// TwinCAT 3 PLC project MCAG_PLC_Project
// ProgramVersion: 3.1.0.8
// libraries:
//   Tc2_MC2, * (Beckhoff Automation GmbH)
//   Tc2_Standard, * (Beckhoff Automation GmbH)
//   Tc2_System, * (Beckhoff Automation GmbH)
//   Tc3_Interfaces, * (Beckhoff Automation GmbH)
//   Tc3_Module, * (Beckhoff Automation GmbH)
// project tree:
//   DUTs/ DUT_AxisStatus_v0_01.TcDUT (not stored), DUT_AxisStatus_v0_02.TcDUT (not stored)
//   / PlcTask.TcTTO (not stored)
//   POUs/Hardware/EtherCAT_Terminals/Analog_Inputs/ FB_CalculateFrequency_3702_v0_01.TcPOU, FB_EL3702_v0_00.TcPOU (not stored), FB_EL3773_v0_00.TcPOU, FB_EL3773_v1_00.TcPOU (not stored)
//   POUs/Hardware/EtherCAT_Terminals/Digital_Inputs/ EL1002_v1_00.TcPOU, EL1004_v1_00.TcPOU (not stored), EL1008_v1_00.TcPOU, EL1012_v1_00.TcPOU (not stored), EL1014_v1_00.TcPOU, EL1018_v1_00.TcPOU, EL1024_v1_00.TcPOU, EL1034_v1_00.TcPOU, EL1084_v1_00.TcPOU (not stored), EL1088_v1_00.TcPOU (not stored), EL1094_v1_00.TcPOU (not stored), EL1098_v1_00.TcPOU, EL1104_v1_00.TcPOU, EL1114_v1_00.TcPOU (not stored), EL1124_v1_00.TcPOU, EL1134_v1_00.TcPOU (not stored), EL1144_v1_00.TcPOU (not stored), EL1202_v1_00.TcPOU, EL1252_v1_00.TcPOU (not stored), EL1258_v0_00.TcPOU, EL1259_v0_00.TcPOU, EL1262_v0_00.TcPOU, EL1502_v0_00.TcPOU (not stored), EL1512_v0_00.TcPOU, EL1702_v1_00.TcPOU, EL1712_v1_00.TcPOU, EL1722_v1_00.TcPOU, EL1804_v1_00.TcPOU (not stored), EL1808_v1_00.TcPOU (not stored), EL1809_v1_00.TcPOU, EL1814_v1_00.TcPOU (not stored), EL1819_v1_00.TcPOU (not stored), EL1859_v1_00.TcPOU (not stored), EL1862_v1_00.TcPOU, EL1872_v1_00.TcPOU (not stored), EL1889_v1_00.TcPOU, FB_EL1008_v1_00.TcPOU (not stored), FB_EL1202_v1_00.TcPOU (not stored), FB_EL1252ASM_v1_00.TcPOU, FB_EL1252_v1_00.TcPOU (not stored)
//   POUs/Hardware/EtherCAT_Terminals/Digital_Outputs/ EL2002_v1_00.TcPOU, EL2004_v1_00.TcPOU (not stored), EL2008_v1_00.TcPOU (not stored), EL2022_v1_00.TcPOU (not stored), EL2024_v1_00.TcPOU (not stored), EL2032_v1_00.TcPOU (not stored), EL2034_v1_00.TcPOU (not stored), EL2042_v1_00.TcPOU, EL2084_v1_00.TcPOU (not stored), EL2088_v1_00.TcPOU (not stored), EL2124_v1_00.TcPOU, EL2202_v0_00.TcPOU, EL2212_v0_00.TcPOU (not stored), EL2252_v0_00.TcPOU, EL2258_v0_00.TcPOU, EL2262_v0_00.TcPOU, EL2502_v0_00.TcPOU (not stored), EL2521_v1_00.TcPOU (not stored), EL2535_v0_00.TcPOU, FB_EL2008_v1_00.TcPOU
//   POUs/Hardware/EtherCAT_Terminals/Digital_Outputs/External_Types/ dutEL2521_Ctrl.TcDUT, dutEL2521_Status.TcDUT
//   POUs/Hardware/EtherCAT_Terminals/Digital_Outputs/Safety_Terminals/ EL1904_v0_00.TcPOU, EL1908_v0_00.TcPOU (not stored), EL2901_v0_00.TcPOU, EL2902_v0_00.TcPOU, EL2904_v0_00.TcPOU (not stored), EL2964_v0_00.TcPOU (not stored), EL6900_v0_00.TcPOU (not stored), FB_EL1904_v1_00.TcPOU (not stored), FB_EL2904_v1_00.TcPOU, FB_EL6900_v1_00.TcPOU
//   POUs/Hardware/EtherCAT_Terminals/Motion/ EL7211_v1_00.TcPOU, EL9576_v1_00.TcPOU
//   POUs/Hardware/EtherCAT_Terminals/System/ EL9505_V1_00.TcPOU
//   POUs/Hardware/Other/ EK1200.TcPOU
//   POUs/ MAIN.TcPOU
//   POUs/Motion/ FB_DriveVirtual.TcPOU, FB_NcAxis.TcPOU (not stored), FB_ReadParameterInNc.TcPOU (not stored), FB_SetPositionBiasInNc_v1_00.TcPOU (not stored), FB_SetPositionBiasInNc.TcPOU (not stored), FB_SetStateToBootstrapOnAX5000.TcPOU (not stored), FB_SetStateToInitOnAX5000.TcPOU (not stored), FB_SimulateEncoder.TcPOU (not stored), FB_WriteParameterInNc.TcPOU (not stored)

// ---- POUs/Hardware/EtherCAT_Terminals/Digital_Outputs/External_Types/dutEL2521_Ctrl.TcDUT
TYPE dutEL2521_Ctrl :
STRUCT
	///The control word (CW) is located in the output process image, and is transmitted from the controller to the terminal.
	///CW.0 FREQ_SEL 0bin / 1bin  Rapid change of the base frequency (only if the ramp function is inactive):
	///0bin = Base frequency 1 (object 8001:02)
	///1bin = Base frequency 2 (object 8001:03) 
	FREQ_SEL: BOOL;
	///CW.1 RAMP_DIS 1bin Operation of the ramp function is cancelled, in spite of object 8000:06 being active; if travel distance control is active, it is interrupted by this bit 
	RAMP_DIS: BOOL;
	///CW.2 GO_COUNTER 1bin  If travel distance control is active (object 8000:0A), then a pre-set counter value is approached when the bit is set 
	GO_COUNTER: BOOL;
	///CW.5 CNT_CLR 1bin The contents of the counter is cleared or set (object 8000:0B) by this bit. 
	///Any overflow or underflow bits that might be set are also cleared by this bit. 
	///The process can be edge triggered or level triggered (object 8000:05). 
	CNT_CLR: BOOL;
END_STRUCT
END_TYPE

// ---- POUs/Hardware/EtherCAT_Terminals/Digital_Outputs/External_Types/dutEL2521_Status.TcDUT
TYPE dutEL2521_Status :
STRUCT
	///The status word (SW) is located in the input process image, and is transmitted from the terminal to the controller.
	///SW.0 SEL_ACK/END_COUNTER 1bin  Confirms the change of base frequency. At activated travel distance control: target counter value reached 
	SEL_ACK: BOOL;
	///SW.1 RAMP_ACTIVE 1bin Ramp is currently being followed 
	RAMP_ACTIVE: BOOL;
	///SW.2 UNDERFLOW 1bin This bit is set if the 16-bit counter underflows (0 -> 65535). It is reset when the counter drops below two thirds of its measuring range (43690 -> 43689) or immediately an overflow occurs. 
	UNDERFLOW: BOOL;
	///SW.3 OVERFLOW 1bin This bit is set if the 16-bit counter overflows (65535 -> 0). It is reset when the counter exceeds one third of its measuring range (21845 -> 21846) or immediately an underflow occurs 
	OVERFLOW: BOOL;
	///SW.4 INPUT_T 1bin Status of INPUT_T 
	INPUT_T: BOOL;
	///SW.5 INPUT_Z 1bin Status of INPUT_Z 
	INPUT_Z: BOOL;
	///SW.6 ERROR 1bin General error bit, included with overflow/underflow 
	ERROR: BOOL;
END_STRUCT
END_TYPE

// ---- POUs/Hardware/EtherCAT_Terminals/Analog_Inputs/FB_CalculateFrequency_3702_v0_01.TcPOU
FUNCTION_BLOCK FB_CalculateFrequency_3702_v0_01
VAR CONSTANT
	///200 samples/period
	cBufferSize: INT := 1000;
END_VAR
VAR_INPUT
	En: BOOL;
	bCalculate: BOOL;
	aBufferValue: ARRAY[0..(cBuffersize - 1)] OF INT;
	aBufferDcTime: ARRAY[0..(cBuffersize - 1)] OF UDINT;
	///If curve has a DC offset
	nDCOffset: INT := 0;
END_VAR
VAR_OUTPUT
	EnO: BOOL;
	bError: BOOL;
	fActFrequency: LREAL;
END_VAR
VAR
	nIndex: INT;
	nFirstZeroCrossing: INT;
	nLastZeroCrossing: INT;
	rTimeFirst: REAL := 0;
	rTimeLast: REAL := 0;
	rTimeRes: REAL := 0;
	nCrossings: INT := 0;
END_VAR
VAR_TEMP
	rRange: REAL := 0;
	rTimeSpan: REAL := 0;
END_VAR

EnO:=En;
bError:=FALSE;
nCrossings:=0;
IF En AND bCalculate THEN
	//Serach for crossings of nDCOffset
	FOR nIndex:=1 TO cBuffersize-1 DO
		IF((aBufferValue[nIndex]>nDCOffset AND aBufferValue[nIndex-1]<=nDCOffset) OR (aBufferValue[nIndex]<nDCOffset AND aBufferValue[nIndex-1]>=nDCOffset))	THEN
			IF(nCrossings=0) THEN
				nFirstZeroCrossing:=nIndex;
			END_IF
			nLastZeroCrossing:=nIndex;
			nCrossings:=nCrossings+1;
		END_IF
	END_FOR	
	
	IF nFirstZeroCrossing < nLastZeroCrossing  AND  nCrossings>2 THEN
		//interpolate zero crossings for higher accuracy
		rTimeRes:=aBufferDcTime[1]-aBufferDcTime[0]; //Buffer must contain more than 2 values
		rRange:=INT_TO_REAL(ABS(aBufferValue[nFirstZeroCrossing-1]-aBufferValue[nFirstZeroCrossing]));
		rTimeFirst:=UDINT_TO_REAL( aBufferDcTime[nFirstZeroCrossing-1])+ABS(INT_TO_REAL(aBufferValue[nFirstZeroCrossing-1])/rRange*rTimeRes);
		rRange:=INT_TO_REAL(ABS(aBufferValue[nLastZeroCrossing-1]-aBufferValue[nLastZeroCrossing]));
		rTimeLast:=UDINT_TO_REAL( aBufferDcTime[nLastZeroCrossing-1])+ABS(INT_TO_REAL(aBufferValue[nLastZeroCrossing-1])/rRange*rTimeRes);

		//Time span first to last (considering that max one time counter overflow have occured in the total time range of the time buffer)	
		IF rTimeFirst<rTimeLast THEN		
			rTimeSpan:=rTimeLast-rTimeFirst;
		ELSE //overflow of counter once (only 32bit timestamp =4.29seconds)
			rTimeSpan:=4294967296.0-rTimeFirst+rTimeLast;
		END_IF
		
		fActFrequency:=1000000000.0/rTimeSpan*(nCrossings-1)/2; //two crossings per period => Average frequency over buffer.
	ELSE
		fActFrequency:=0;
	END_IF
END_IF

END_FUNCTION_BLOCK

// ---- POUs/Hardware/EtherCAT_Terminals/Analog_Inputs/FB_EL3773_v0_00.TcPOU
FUNCTION_BLOCK FB_EL3773_v0_00
VAR_INPUT
	En: BOOL;
END_VAR
VAR_OUTPUT
	EnO: BOOL;
	bL1Ok: BOOL;
	aL1Voltage: ARRAY[0..(cDcOversampling - 1)] OF INT;
	aL1Current: ARRAY[0..(cDcOversampling - 1)] OF INT;
	bL2Ok: BOOL;
	aL2Voltage: ARRAY[0..(cDcOversampling - 1)] OF INT;
	aL2Current: ARRAY[0..(cDcOversampling - 1)] OF INT;
	bL3Ok: BOOL;
	aL3Voltage: ARRAY[0..(cDcOversampling - 1)] OF INT;
	aL3Current: ARRAY[0..(cDcOversampling - 1)] OF INT;
	nDcTimeNextLatch: ULINT;
	bError: BOOL;
END_VAR
VAR
	L1_Voltage_Status_U1 AT %I*: UINT;
	L1_Voltage_Samples_U1_Samples AT %I*: ARRAY[0..(cDcOversampling - 1)] OF INT;
	L1_Current_Status_I1_Status AT %I*: UINT;
	L1_Current_Samples_I1_Samples AT %I*: ARRAY[0..(cDcOversampling - 1)] OF INT;
	L2_Voltage_Status_U2 AT %I*: UINT;
	L2_Voltage_Samples_U2_Samples AT %I*: ARRAY[0..(cDcOversampling - 1)] OF INT;
	L2_Current_Status_I2_Status AT %I*: UINT;
	L2_Current_Samples_I2_Samples AT %I*: ARRAY[0..(cDcOversampling - 1)] OF INT;
	L3_Voltage_Status_U3 AT %I*: UINT;
	L3_Voltage_Samples_U3_Samples AT %I*: ARRAY[0..(cDcOversampling - 1)] OF INT;
	L3_Current_Status_I3_Status AT %I*: UINT;
	L3_Current_Samples_I3_Samples AT %I*: ARRAY[0..(cDcOversampling - 1)] OF INT;
	AI_NextSync1Time_StartTimeNextLatch AT %I*: ULINT;
	WcState_WcState AT %I*: BOOL;
	InfoData_State AT %I*: UINT;
END_VAR

EnO:=En;

IF En AND (WcState_WcState OR InfoData_State<>16#8) THEN
	bError:=TRUE;
ELSE
	bError:=FALSE;
END_IF


IF En THEN
	IF bError=FALSE THEN
		IF (L1_Voltage_Status_U1 AND 2#0110000001000011)<>0
		OR (L1_Current_Status_I1_Status AND 2#0110000001000011)<>0 THEN
			bL1Ok:= FALSE;
		ELSE
			bL1Ok:= TRUE;
		END_IF
		
		IF (L2_Voltage_Status_U2 AND 2#0110000001000011)<>0
		OR (L2_Current_Status_I2_Status AND 2#0110000001000011)<>0 THEN
			bL2Ok:= FALSE;
		ELSE
			bL2Ok:= TRUE;
		END_IF
		
		IF (L3_Voltage_Status_U3 AND 2#0110000001000011)<>0
		OR (L3_Current_Status_I3_Status AND 2#0110000001000011)<>0 THEN
			bL3Ok:= FALSE;
		ELSE
			bL3Ok:= TRUE;
		END_IF

		IF bL1Ok THEN
			aL1Voltage:=L1_Voltage_Samples_U1_Samples;
			aL1Current:=L1_Current_Samples_I1_Samples;
		END_IF

		IF bL2Ok THEN
			aL2Voltage:=L2_Voltage_Samples_U2_Samples;
			aL2Current:=L2_Current_Samples_I2_Samples;
		END_IF

		IF bL3Ok THEN
			aL3Voltage:=L3_Voltage_Samples_U3_Samples;
			aL3Current:=L3_Current_Samples_I3_Samples;
		END_IF

		nDcTimeNextLatch:=AI_NextSync1Time_StartTimeNextLatch;
	ELSE
		bL1Ok:= FALSE;
		bL2Ok:= FALSE;
		bL3Ok:= FALSE;
		nDcTimeNextLatch:=0;
	END_IF
END_IF

END_FUNCTION_BLOCK

// ---- POUs/Hardware/EtherCAT_Terminals/Digital_Inputs/EL1002_v1_00.TcPOU
///EL1002 | 2-channel digital input terminal 24 V DC, 3 ms
FUNCTION_BLOCK EL1002_v1_00
VAR_INPUT
	En: BOOL;
END_VAR
VAR_OUTPUT
	EnO: BOOL;
	bDi_1: BOOL;
	bDi_2: BOOL;
	bError: BOOL;
END_VAR
VAR
	Channel_1_Input AT %I*: BOOL;
	Channel_2_Input AT %I*: BOOL;
	WcState_WcState AT %I*: BOOL;
	InfoData_State AT %I*: UINT;
END_VAR

EnO:=En;

IF En AND (WcState_WcState OR InfoData_State<>16#8) THEN
	bError:=TRUE;
ELSE
	bError:=FALSE;
END_IF

IF En THEN
	IF bError=FALSE THEN
		bDi_1:=Channel_1_Input;
		bDi_2:=Channel_2_Input;
	ELSE
		bDi_1:=FALSE;
		bDi_2:=FALSE;
	END_IF
END_IF

END_FUNCTION_BLOCK

// ---- POUs/Hardware/EtherCAT_Terminals/Digital_Inputs/EL1008_v1_00.TcPOU
///EL1008 | 8-channel digital input terminal 24 V DC, 3 ms
FUNCTION_BLOCK EL1008_v1_00
VAR_INPUT
	En: BOOL;
END_VAR
VAR_OUTPUT
	EnO: BOOL;
	bDi_1: BOOL;
	bDi_2: BOOL;
	bDi_3: BOOL;
	bDi_4: BOOL;
	bDi_5: BOOL;
	bDi_6: BOOL;
	bDi_7: BOOL;
	bDi_8: BOOL;
	bError: BOOL;
END_VAR
VAR
	Channel_1_Input AT %I*: BOOL;
	Channel_2_Input AT %I*: BOOL;
	Channel_3_Input AT %I*: BOOL;
	Channel_4_Input AT %I*: BOOL;
	Channel_5_Input AT %I*: BOOL;
	Channel_6_Input AT %I*: BOOL;
	Channel_7_Input AT %I*: BOOL;
	Channel_8_Input AT %I*: BOOL;
	WcState_WcState AT %I*: BOOL;
	InfoData_State AT %I*: UINT;
END_VAR

EnO:=En;

IF En AND (WcState_WcState OR InfoData_State<>16#8) THEN
	bError:=TRUE;
ELSE
	bError:=FALSE;
END_IF

IF En THEN
	IF bError=FALSE THEN
		bDi_1:=Channel_1_Input;
		bDi_2:=Channel_2_Input;
		bDi_3:=Channel_3_Input;
		bDi_4:=Channel_4_Input;
		bDi_5:=Channel_5_Input;
		bDi_6:=Channel_6_Input;
		bDi_7:=Channel_7_Input;
		bDi_8:=Channel_8_Input;
	ELSE
		bDi_1:=FALSE;
		bDi_2:=FALSE;
		bDi_3:=FALSE;
		bDi_4:=FALSE;
		bDi_5:=FALSE;
		bDi_6:=FALSE;
		bDi_7:=FALSE;
		bDi_8:=FALSE;
	END_IF
END_IF

END_FUNCTION_BLOCK

// ---- POUs/Hardware/EtherCAT_Terminals/Digital_Inputs/EL1014_v1_00.TcPOU
///EL1014 | 4-channel digital input terminal 24 V DC, 10 µs
FUNCTION_BLOCK EL1014_v1_00
VAR_INPUT
	En: BOOL;
END_VAR
VAR_OUTPUT
	EnO: BOOL;
	bDi_1: BOOL;
	bDi_2: BOOL;
	bDi_3: BOOL;
	bDi_4: BOOL;
	bError: BOOL;
END_VAR
VAR
	Channel_1_Input AT %I*: BOOL;
	Channel_2_Input AT %I*: BOOL;
	Channel_3_Input AT %I*: BOOL;
	Channel_4_Input AT %I*: BOOL;
	WcState_WcState AT %I*: BOOL;
	InfoData_State AT %I*: UINT;
END_VAR

EnO:=En;

IF En AND (WcState_WcState OR InfoData_State<>16#8) THEN
	bError:=TRUE;
ELSE
	bError:=FALSE;
END_IF

IF En THEN
	IF bError=FALSE THEN
		bDi_1:=Channel_1_Input;
		bDi_2:=Channel_2_Input;
		bDi_3:=Channel_3_Input;
		bDi_4:=Channel_4_Input;
	ELSE
		bDi_1:=FALSE;
		bDi_2:=FALSE;
		bDi_3:=FALSE;
		bDi_4:=FALSE;
	END_IF
END_IF

END_FUNCTION_BLOCK

// ---- POUs/Hardware/EtherCAT_Terminals/Digital_Inputs/EL1018_v1_00.TcPOU
///EL1018 | 8-channel digital input terminal 24 V DC, 10 µs
FUNCTION_BLOCK EL1018_v1_00
VAR_INPUT
	En: BOOL;
END_VAR
VAR_OUTPUT
	EnO: BOOL;
	bDi_1: BOOL;
	bDi_2: BOOL;
	bDi_3: BOOL;
	bDi_4: BOOL;
	bDi_5: BOOL;
	bDi_6: BOOL;
	bDi_7: BOOL;
	bDi_8: BOOL;
	bError: BOOL;
END_VAR
VAR
	Channel_1_Input AT %I*: BOOL;
	Channel_2_Input AT %I*: BOOL;
	Channel_3_Input AT %I*: BOOL;
	Channel_4_Input AT %I*: BOOL;
	Channel_5_Input AT %I*: BOOL;
	Channel_6_Input AT %I*: BOOL;
	Channel_7_Input AT %I*: BOOL;
	Channel_8_Input AT %I*: BOOL;
	WcState_WcState AT %I*: BOOL;
	InfoData_State AT %I*: UINT;
END_VAR

EnO:=En;

IF En AND (WcState_WcState OR InfoData_State<>16#8) THEN
	bError:=TRUE;
ELSE
	bError:=FALSE;
END_IF

IF En THEN
	IF bError=FALSE THEN
		bDi_1:=Channel_1_Input;
		bDi_2:=Channel_2_Input;
		bDi_3:=Channel_3_Input;
		bDi_4:=Channel_4_Input;
		bDi_5:=Channel_5_Input;
		bDi_6:=Channel_6_Input;
		bDi_7:=Channel_7_Input;
		bDi_8:=Channel_8_Input;
	ELSE
		bDi_1:=FALSE;
		bDi_2:=FALSE;
		bDi_3:=FALSE;
		bDi_4:=FALSE;
		bDi_5:=FALSE;
		bDi_6:=FALSE;
		bDi_7:=FALSE;
		bDi_8:=FALSE;
	END_IF
END_IF

END_FUNCTION_BLOCK

// ---- POUs/Hardware/EtherCAT_Terminals/Digital_Inputs/EL1024_v1_00.TcPOU
///EL1024 | 4-channel digital input terminal 24 V DC, 3 ms, for type 2 sensors
FUNCTION_BLOCK EL1024_v1_00
VAR_INPUT
	En: BOOL;
END_VAR
VAR_OUTPUT
	EnO: BOOL;
	bDi_1: BOOL;
	bDi_2: BOOL;
	bDi_3: BOOL;
	bDi_4: BOOL;
	bError: BOOL;
END_VAR
VAR
	Channel_1_Input AT %I*: BOOL;
	Channel_2_Input AT %I*: BOOL;
	Channel_3_Input AT %I*: BOOL;
	Channel_4_Input AT %I*: BOOL;
	WcState_WcState AT %I*: BOOL;
	InfoData_State AT %I*: UINT;
END_VAR

EnO:=En;

IF En AND (WcState_WcState OR InfoData_State<>16#8) THEN
	bError:=TRUE;
ELSE
	bError:=FALSE;
END_IF

IF En THEN
	IF bError=FALSE THEN
		bDi_1:=Channel_1_Input;
		bDi_2:=Channel_2_Input;
		bDi_3:=Channel_3_Input;
		bDi_4:=Channel_4_Input;
	ELSE
		bDi_1:=FALSE;
		bDi_2:=FALSE;
		bDi_3:=FALSE;
		bDi_4:=FALSE;
	END_IF
END_IF

END_FUNCTION_BLOCK

// ---- POUs/Hardware/EtherCAT_Terminals/Digital_Inputs/EL1034_v1_00.TcPOU
///EL1034 | 4-channel digital input terminal 24 V DC, 10 µs, potential-free inputs
FUNCTION_BLOCK EL1034_v1_00
VAR_INPUT
	En: BOOL;
END_VAR
VAR_OUTPUT
	EnO: BOOL;
	bDi_1: BOOL;
	bDi_2: BOOL;
	bDi_3: BOOL;
	bDi_4: BOOL;
	bError: BOOL;
END_VAR
VAR
	Channel_1_Input AT %I*: BOOL;
	Channel_2_Input AT %I*: BOOL;
	Channel_3_Input AT %I*: BOOL;
	Channel_4_Input AT %I*: BOOL;
	WcState_WcState AT %I*: BOOL;
	InfoData_State AT %I*: UINT;
END_VAR

EnO:=En;

IF En AND (WcState_WcState OR InfoData_State<>16#8) THEN
	bError:=TRUE;
ELSE
	bError:=FALSE;
END_IF

IF En THEN
	IF bError=FALSE THEN
		bDi_1:=Channel_1_Input;
		bDi_2:=Channel_2_Input;
		bDi_3:=Channel_3_Input;
		bDi_4:=Channel_4_Input;
	ELSE
		bDi_1:=FALSE;
		bDi_2:=FALSE;
		bDi_3:=FALSE;
		bDi_4:=FALSE;
	END_IF
END_IF

END_FUNCTION_BLOCK

// ---- POUs/Hardware/EtherCAT_Terminals/Digital_Inputs/EL1098_v1_00.TcPOU
///EL1098 | 8-channel digital input terminal 24 V DC, 10 µs, switching to negative potential
FUNCTION_BLOCK EL1098_v1_00
VAR_INPUT
	En: BOOL;
END_VAR
VAR_OUTPUT
	EnO: BOOL;
	bDi_1: BOOL;
	bDi_2: BOOL;
	bDi_3: BOOL;
	bDi_4: BOOL;
	bDi_5: BOOL;
	bDi_6: BOOL;
	bDi_7: BOOL;
	bDi_8: BOOL;
	bError: BOOL;
END_VAR
VAR
	Channel_1_Input AT %I*: BOOL;
	Channel_2_Input AT %I*: BOOL;
	Channel_3_Input AT %I*: BOOL;
	Channel_4_Input AT %I*: BOOL;
	Channel_5_Input AT %I*: BOOL;
	Channel_6_Input AT %I*: BOOL;
	Channel_7_Input AT %I*: BOOL;
	Channel_8_Input AT %I*: BOOL;
	WcState_WcState AT %I*: BOOL;
	InfoData_State AT %I*: UINT;
END_VAR

EnO:=En;

IF En AND (WcState_WcState OR InfoData_State<>16#8) THEN
	bError:=TRUE;
ELSE
	bError:=FALSE;
END_IF

IF En THEN
	IF bError=FALSE THEN
		bDi_1:=Channel_1_Input;
		bDi_2:=Channel_2_Input;
		bDi_3:=Channel_3_Input;
		bDi_4:=Channel_4_Input;
		bDi_5:=Channel_5_Input;
		bDi_6:=Channel_6_Input;
		bDi_7:=Channel_7_Input;
		bDi_8:=Channel_8_Input;
	ELSE
		bDi_1:=FALSE;
		bDi_2:=FALSE;
		bDi_3:=FALSE;
		bDi_4:=FALSE;
		bDi_5:=FALSE;
		bDi_6:=FALSE;
		bDi_7:=FALSE;
		bDi_8:=FALSE;
	END_IF
END_IF

END_FUNCTION_BLOCK

// ---- POUs/Hardware/EtherCAT_Terminals/Digital_Inputs/EL1104_v1_00.TcPOU
///EL1104 | 4-channel digital input terminals 24 V DC, 3 ms, 24 V and 0 V sensor supply
FUNCTION_BLOCK EL1104_v1_00
VAR_INPUT
	En: BOOL;
END_VAR
VAR_OUTPUT
	EnO: BOOL;
	bDi_1: BOOL;
	bDi_2: BOOL;
	bDi_3: BOOL;
	bDi_4: BOOL;
	bError: BOOL;
END_VAR
VAR
	Channel_1_Input AT %I*: BOOL;
	Channel_2_Input AT %I*: BOOL;
	Channel_3_Input AT %I*: BOOL;
	Channel_4_Input AT %I*: BOOL;
	WcState_WcState AT %I*: BOOL;
	InfoData_State AT %I*: UINT;
END_VAR

EnO:=En;

IF En AND (WcState_WcState OR InfoData_State<>16#8) THEN
	bError:=TRUE;
ELSE
	bError:=FALSE;
END_IF

IF En THEN
	IF bError=FALSE THEN
		bDi_1:=Channel_1_Input;
		bDi_2:=Channel_2_Input;
		bDi_3:=Channel_3_Input;
		bDi_4:=Channel_4_Input;
	ELSE
		bDi_1:=FALSE;
		bDi_2:=FALSE;
		bDi_3:=FALSE;
		bDi_4:=FALSE;
	END_IF
END_IF

END_FUNCTION_BLOCK

// ---- POUs/Hardware/EtherCAT_Terminals/Digital_Inputs/EL1124_v1_00.TcPOU
///EL1124 | 4-channel digital input terminal 5 V DC, 0.5 µs
FUNCTION_BLOCK EL1124_v1_00
VAR_INPUT
	En: BOOL;
END_VAR
VAR_OUTPUT
	EnO: BOOL;
	bDi_1: BOOL;
	bDi_2: BOOL;
	bDi_3: BOOL;
	bDi_4: BOOL;
	bError: BOOL;
END_VAR
VAR
	Channel_1_Input AT %I*: BOOL;
	Channel_2_Input AT %I*: BOOL;
	Channel_3_Input AT %I*: BOOL;
	Channel_4_Input AT %I*: BOOL;
	WcState_WcState AT %I*: BOOL;
	InfoData_State AT %I*: UINT;
END_VAR

EnO:=En;

IF En AND (WcState_WcState OR InfoData_State<>16#8) THEN
	bError:=TRUE;
ELSE
	bError:=FALSE;
END_IF

IF En THEN
	IF bError=FALSE THEN
		bDi_1:=Channel_1_Input;
		bDi_2:=Channel_2_Input;
		bDi_3:=Channel_3_Input;
		bDi_4:=Channel_4_Input;
	ELSE
		bDi_1:=FALSE;
		bDi_2:=FALSE;
		bDi_3:=FALSE;
		bDi_4:=FALSE;
	END_IF
END_IF

END_FUNCTION_BLOCK

// ---- POUs/Hardware/EtherCAT_Terminals/Digital_Inputs/EL1202_v1_00.TcPOU
///EL1202 | XFC, 2-channel digital input terminal 24 V DC, TON/TOFF 1 µs
FUNCTION_BLOCK EL1202_v1_00
VAR_INPUT
	En: BOOL;
END_VAR
VAR_OUTPUT
	EnO: BOOL;
	bDi_1: BOOL;
	bDi_2: BOOL;
	bError: BOOL;
END_VAR
VAR
	Channel_1_Input AT %I*: BOOL;
	Channel_2_Input AT %I*: BOOL;
	WcState_WcState AT %I*: BOOL;
	InfoData_State AT %I*: UINT;
END_VAR

EnO:=En;

IF En AND (WcState_WcState OR InfoData_State<>16#8) THEN
	bError:=TRUE;
ELSE
	bError:=FALSE;
END_IF

IF En THEN
	IF bError=FALSE THEN
		bDi_1:=Channel_1_Input;
		bDi_2:=Channel_2_Input;
	ELSE
		bDi_1:=FALSE;
		bDi_2:=FALSE;
	END_IF
END_IF

END_FUNCTION_BLOCK

// ---- POUs/Hardware/EtherCAT_Terminals/Digital_Inputs/EL1258_v0_00.TcPOU
///EL1258 | XFC, 8-channel digital input terminal with time stamp
FUNCTION_BLOCK EL1258_v0_00

END_FUNCTION_BLOCK

// ---- POUs/Hardware/EtherCAT_Terminals/Digital_Inputs/EL1259_v0_00.TcPOU
///EL1259 | XFC, 8-channel digital input + 8-channel digital output with Time-Stamp
FUNCTION_BLOCK EL1259_v0_00

END_FUNCTION_BLOCK

// ---- POUs/Hardware/EtherCAT_Terminals/Digital_Inputs/EL1262_v0_00.TcPOU
///EL1262 | XFC, 2-channel digital input terminal with oversampling
FUNCTION_BLOCK EL1262_v0_00

END_FUNCTION_BLOCK

// ---- POUs/Hardware/EtherCAT_Terminals/Digital_Inputs/EL1512_v0_00.TcPOU
///EL1512 | 2-channel, up/down counter, 24 V DC, 1 kHz, 16 bit
FUNCTION_BLOCK EL1512_v0_00

END_FUNCTION_BLOCK

// ---- POUs/Hardware/EtherCAT_Terminals/Digital_Inputs/EL1702_v1_00.TcPOU
///EL1702 | 2-channel digital input terminals 120V/230V AC, 10ms
FUNCTION_BLOCK EL1702_v1_00
VAR_INPUT
	En: BOOL;
END_VAR
VAR_OUTPUT
	EnO: BOOL;
	bDi_1: BOOL;
	bDi_2: BOOL;
	bError: BOOL;
END_VAR
VAR
	Channel_1_Input AT %I*: BOOL;
	Channel_2_Input AT %I*: BOOL;
	WcState_WcState AT %I*: BOOL;
	InfoData_State AT %I*: UINT;
END_VAR

EnO:=En;

IF En AND (WcState_WcState OR InfoData_State<>16#8) THEN
	bError:=TRUE;
ELSE
	bError:=FALSE;
END_IF

IF En THEN
	IF bError=FALSE THEN
		bDi_1:=Channel_1_Input;
		bDi_2:=Channel_2_Input;
	ELSE
		bDi_1:=FALSE;
		bDi_2:=FALSE;
	END_IF
END_IF

END_FUNCTION_BLOCK

// ---- POUs/Hardware/EtherCAT_Terminals/Digital_Inputs/EL1712_v1_00.TcPOU
///EL1712 | 2-channel digital input terminals 120V AC/DC, 10ms
FUNCTION_BLOCK EL1712_v1_00
VAR_INPUT
	En: BOOL;
END_VAR
VAR_OUTPUT
	EnO: BOOL;
	bDi_1: BOOL;
	bDi_2: BOOL;
	bError: BOOL;
END_VAR
VAR
	Channel_1_Input AT %I*: BOOL;
	Channel_2_Input AT %I*: BOOL;
	WcState_WcState AT %I*: BOOL;
	InfoData_State AT %I*: UINT;
END_VAR

EnO:=En;

IF En AND (WcState_WcState OR InfoData_State<>16#8) THEN
	bError:=TRUE;
ELSE
	bError:=FALSE;
END_IF

IF En THEN
	IF bError=FALSE THEN
		bDi_1:=Channel_1_Input;
		bDi_2:=Channel_2_Input;
	ELSE
		bDi_1:=FALSE;
		bDi_2:=FALSE;
	END_IF
END_IF

END_FUNCTION_BLOCK

// ---- POUs/Hardware/EtherCAT_Terminals/Digital_Inputs/EL1722_v1_00.TcPOU
///EL1722 | 2-channel digital input terminals 120V/230V AC, 10ms, no power contacts
FUNCTION_BLOCK EL1722_v1_00
VAR_INPUT
	En: BOOL;
END_VAR
VAR_OUTPUT
	EnO: BOOL;
	bDi_1: BOOL;
	bDi_2: BOOL;
	bError: BOOL;
END_VAR
VAR
	Channel_1_Input AT %I*: BOOL;
	Channel_2_Input AT %I*: BOOL;
	WcState_WcState AT %I*: BOOL;
	InfoData_State AT %I*: UINT;
END_VAR

EnO:=En;

IF En AND (WcState_WcState OR InfoData_State<>16#8) THEN
	bError:=TRUE;
ELSE
	bError:=FALSE;
END_IF

IF En THEN
	IF bError=FALSE THEN
		bDi_1:=Channel_1_Input;
		bDi_2:=Channel_2_Input;
	ELSE
		bDi_1:=FALSE;
		bDi_2:=FALSE;
	END_IF
END_IF

END_FUNCTION_BLOCK

// ---- POUs/Hardware/EtherCAT_Terminals/Digital_Inputs/EL1809_v1_00.TcPOU
///EL1809 | HD EtherCAT Terminals, 16-channel digital input 24 V DC, 3 ms
FUNCTION_BLOCK EL1809_v1_00
VAR_INPUT
	En: BOOL;
END_VAR
VAR_OUTPUT
	EnO: BOOL;
	bDi_1: BOOL;
	bDi_2: BOOL;
	bDi_3: BOOL;
	bDi_4: BOOL;
	bDi_5: BOOL;
	bDi_6: BOOL;
	bDi_7: BOOL;
	bDi_8: BOOL;
	bDi_9: BOOL;
	bDi_10: BOOL;
	bDi_11: BOOL;
	bDi_12: BOOL;
	bDi_13: BOOL;
	bDi_14: BOOL;
	bDi_15: BOOL;
	bDi_16: BOOL;
	bError: BOOL;
END_VAR
VAR
	Channel_1_Input AT %I*: BOOL;
	Channel_2_Input AT %I*: BOOL;
	Channel_3_Input AT %I*: BOOL;
	Channel_4_Input AT %I*: BOOL;
	Channel_5_Input AT %I*: BOOL;
	Channel_6_Input AT %I*: BOOL;
	Channel_7_Input AT %I*: BOOL;
	Channel_8_Input AT %I*: BOOL;
	Channel_9_Input AT %I*: BOOL;
	Channel_10_Input AT %I*: BOOL;
	Channel_11_Input AT %I*: BOOL;
	Channel_12_Input AT %I*: BOOL;
	Channel_13_Input AT %I*: BOOL;
	Channel_14_Input AT %I*: BOOL;
	Channel_15_Input AT %I*: BOOL;
	Channel_16_Input AT %I*: BOOL;
	WcState_WcState AT %I*: BOOL;
	InfoData_State AT %I*: UINT;
END_VAR

EnO:=En;

IF En AND (WcState_WcState OR InfoData_State<>16#8) THEN
	bError:=TRUE;
ELSE
	bError:=FALSE;
END_IF

IF En THEN
	IF bError=FALSE THEN
		bDi_1:=Channel_1_Input;
		bDi_2:=Channel_2_Input;
		bDi_3:=Channel_3_Input;
		bDi_4:=Channel_4_Input;
		bDi_5:=Channel_5_Input;
		bDi_6:=Channel_6_Input;
		bDi_7:=Channel_7_Input;
		bDi_8:=Channel_8_Input;
		bDi_9:=Channel_9_Input;
		bDi_10:=Channel_10_Input;
		bDi_11:=Channel_11_Input;
		bDi_12:=Channel_12_Input;
		bDi_13:=Channel_13_Input;
		bDi_14:=Channel_14_Input;
		bDi_15:=Channel_15_Input;
		bDi_16:=Channel_16_Input;
	ELSE
		bDi_1:=FALSE;
		bDi_2:=FALSE;
		bDi_3:=FALSE;
		bDi_4:=FALSE;
		bDi_5:=FALSE;
		bDi_6:=FALSE;
		bDi_7:=FALSE;
		bDi_8:=FALSE;
		bDi_9:=FALSE;
		bDi_10:=FALSE;
		bDi_11:=FALSE;
		bDi_12:=FALSE;
		bDi_13:=FALSE;
		bDi_14:=FALSE;
		bDi_15:=FALSE;
		bDi_16:=FALSE;
	END_IF
END_IF

END_FUNCTION_BLOCK

// ---- POUs/Hardware/EtherCAT_Terminals/Digital_Inputs/EL1862_v1_00.TcPOU
///EL1862 | 16-channel digital input terminals 24 V DC, 3 ms, type 3, flat-ribbon cable connection
FUNCTION_BLOCK EL1862_v1_00
VAR_INPUT
	En: BOOL;
END_VAR
VAR_OUTPUT
	EnO: BOOL;
	bDi_1: BOOL;
	bDi_2: BOOL;
	bDi_3: BOOL;
	bDi_4: BOOL;
	bDi_5: BOOL;
	bDi_6: BOOL;
	bDi_7: BOOL;
	bDi_8: BOOL;
	bDi_9: BOOL;
	bDi_10: BOOL;
	bDi_11: BOOL;
	bDi_12: BOOL;
	bDi_13: BOOL;
	bDi_14: BOOL;
	bDi_15: BOOL;
	bDi_16: BOOL;
	bError: BOOL;
END_VAR
VAR
	Channel_1_Input AT %I*: BOOL;
	Channel_2_Input AT %I*: BOOL;
	Channel_3_Input AT %I*: BOOL;
	Channel_4_Input AT %I*: BOOL;
	Channel_5_Input AT %I*: BOOL;
	Channel_6_Input AT %I*: BOOL;
	Channel_7_Input AT %I*: BOOL;
	Channel_8_Input AT %I*: BOOL;
	Channel_9_Input AT %I*: BOOL;
	Channel_10_Input AT %I*: BOOL;
	Channel_11_Input AT %I*: BOOL;
	Channel_12_Input AT %I*: BOOL;
	Channel_13_Input AT %I*: BOOL;
	Channel_14_Input AT %I*: BOOL;
	Channel_15_Input AT %I*: BOOL;
	Channel_16_Input AT %I*: BOOL;
	WcState_WcState AT %I*: BOOL;
	InfoData_State AT %I*: UINT;
END_VAR

EnO:=En;

IF En AND (WcState_WcState OR InfoData_State<>16#8) THEN
	bError:=TRUE;
ELSE
	bError:=FALSE;
END_IF

IF En THEN
	IF bError=FALSE THEN
		bDi_1:=Channel_1_Input;
		bDi_2:=Channel_2_Input;
		bDi_3:=Channel_3_Input;
		bDi_4:=Channel_4_Input;
		bDi_5:=Channel_5_Input;
		bDi_6:=Channel_6_Input;
		bDi_7:=Channel_7_Input;
		bDi_8:=Channel_8_Input;
		bDi_9:=Channel_9_Input;
		bDi_10:=Channel_10_Input;
		bDi_11:=Channel_11_Input;
		bDi_12:=Channel_12_Input;
		bDi_13:=Channel_13_Input;
		bDi_14:=Channel_14_Input;
		bDi_15:=Channel_15_Input;
		bDi_16:=Channel_16_Input;
	ELSE
		bDi_1:=FALSE;
		bDi_2:=FALSE;
		bDi_3:=FALSE;
		bDi_4:=FALSE;
		bDi_5:=FALSE;
		bDi_6:=FALSE;
		bDi_7:=FALSE;
		bDi_8:=FALSE;
		bDi_9:=FALSE;
		bDi_10:=FALSE;
		bDi_11:=FALSE;
		bDi_12:=FALSE;
		bDi_13:=FALSE;
		bDi_14:=FALSE;
		bDi_15:=FALSE;
		bDi_16:=FALSE;
	END_IF
END_IF

END_FUNCTION_BLOCK

// ---- POUs/Hardware/EtherCAT_Terminals/Digital_Inputs/EL1889_v1_00.TcPOU
///EL1889 | HD EtherCAT Terminal, 16-channel digital input 24 V DC, 3 ms, 0 V (ground) switching
FUNCTION_BLOCK EL1889_v1_00
VAR_INPUT
	En: BOOL;
END_VAR
VAR_OUTPUT
	EnO: BOOL;
	bDi_1: BOOL;
	bDi_2: BOOL;
	bDi_3: BOOL;
	bDi_4: BOOL;
	bDi_5: BOOL;
	bDi_6: BOOL;
	bDi_7: BOOL;
	bDi_8: BOOL;
	bDi_9: BOOL;
	bDi_10: BOOL;
	bDi_11: BOOL;
	bDi_12: BOOL;
	bDi_13: BOOL;
	bDi_14: BOOL;
	bDi_15: BOOL;
	bDi_16: BOOL;
	bError: BOOL;
END_VAR
VAR
	Channel_1_Input AT %I*: BOOL;
	Channel_2_Input AT %I*: BOOL;
	Channel_3_Input AT %I*: BOOL;
	Channel_4_Input AT %I*: BOOL;
	Channel_5_Input AT %I*: BOOL;
	Channel_6_Input AT %I*: BOOL;
	Channel_7_Input AT %I*: BOOL;
	Channel_8_Input AT %I*: BOOL;
	Channel_9_Input AT %I*: BOOL;
	Channel_10_Input AT %I*: BOOL;
	Channel_11_Input AT %I*: BOOL;
	Channel_12_Input AT %I*: BOOL;
	Channel_13_Input AT %I*: BOOL;
	Channel_14_Input AT %I*: BOOL;
	Channel_15_Input AT %I*: BOOL;
	Channel_16_Input AT %I*: BOOL;
	WcState_WcState AT %I*: BOOL;
	InfoData_State AT %I*: UINT;
END_VAR

EnO:=En;

IF En AND (WcState_WcState OR InfoData_State<>16#8) THEN
	bError:=TRUE;
ELSE
	bError:=FALSE;
END_IF

IF En THEN
	IF bError=FALSE THEN
		bDi_1:=Channel_1_Input;
		bDi_2:=Channel_2_Input;
		bDi_3:=Channel_3_Input;
		bDi_4:=Channel_4_Input;
		bDi_5:=Channel_5_Input;
		bDi_6:=Channel_6_Input;
		bDi_7:=Channel_7_Input;
		bDi_8:=Channel_8_Input;
		bDi_9:=Channel_9_Input;
		bDi_10:=Channel_10_Input;
		bDi_11:=Channel_11_Input;
		bDi_12:=Channel_12_Input;
		bDi_13:=Channel_13_Input;
		bDi_14:=Channel_14_Input;
		bDi_15:=Channel_15_Input;
		bDi_16:=Channel_16_Input;
	ELSE
		bDi_1:=FALSE;
		bDi_2:=FALSE;
		bDi_3:=FALSE;
		bDi_4:=FALSE;
		bDi_5:=FALSE;
		bDi_6:=FALSE;
		bDi_7:=FALSE;
		bDi_8:=FALSE;
		bDi_9:=FALSE;
		bDi_10:=FALSE;
		bDi_11:=FALSE;
		bDi_12:=FALSE;
		bDi_13:=FALSE;
		bDi_14:=FALSE;
		bDi_15:=FALSE;
		bDi_16:=FALSE;
	END_IF
END_IF

END_FUNCTION_BLOCK

// ---- POUs/Hardware/EtherCAT_Terminals/Digital_Inputs/FB_EL1252ASM_v1_00.TcPOU
FUNCTION_BLOCK FB_EL1252ASM_v1_00
VAR_INPUT
	En: BOOL;
END_VAR
VAR_OUTPUT
	EnO: BOOL;
	Di_1: BOOL;
	Di_2: BOOL;
	Di_1_LatchTimePos: ULINT;
	Di_2_LatchTimePos: ULINT;
	Di_1_LatchTimeNeg: ULINT;
	Di_2_LatchTimeNeg: ULINT;
	///Below bits can be used but then they must be enabled in the COE of the card. Nicklas suggested to not use these (since something wss written that you then only were allowed to read the latch time onece (some kkind of auto reset??))	
	///Di_1_LatchNeg:BOOL;
	///	Di_1_LatchPos:BOOL;
	///	Di_2_LatchNeg:BOOL;
	///	Di_2_LatchPos:BOOL;
	Error: BOOL;
END_VAR
VAR
	Channel_1_Input AT %I*: BOOL;
	Channel_2_Input AT %I*: BOOL;
	///Latch_Status1 AT %I*: USINT;
	///	Latch_Status2 AT %I*: USINT;
	Latch_LatchPos1 AT %I*: ULINT;
	Latch_LatchNeg1 AT %I*: ULINT;
	Latch_LatchPos2 AT %I*: ULINT;
	Latch_LatchNeg2 AT %I*: ULINT;
	WcState_WcState AT %I*: BOOL;
	InfoData_State AT %I*: UINT;
END_VAR

EnO:=En;

IF En AND (WcState_WcState OR InfoData_State<>16#8) THEN //InfoData_State==0 => in OP mode
	Error:=TRUE;
ELSE
	Error:=FALSE;
END_IF

IF En THEN
	IF Error=FALSE THEN
		Di_1:=Channel_1_Input;
		Di_2:=Channel_2_Input;
	(*	Di_1_LatchPos:=Latch_Status1.0;
		Di_1_LatchNeg:=Latch_Status1.1;
		Di_2_LatchPos:=Latch_Status2.0;
		Di_2_LatchNeg:=Latch_Status2.1;*)
		Di_1_LatchTimePos:=Latch_LatchPos1;
		Di_2_LatchTimePos:=Latch_LatchPos2;		
		Di_1_LatchTimeNeg:=Latch_LatchNeg1;		
		Di_2_LatchTimeNeg:=Latch_LatchNeg2;
		
	ELSE
		Di_1:=FALSE;
		Di_2:=FALSE;
	END_IF
END_IF

END_FUNCTION_BLOCK

// ---- POUs/Hardware/EtherCAT_Terminals/Digital_Outputs/EL2002_v1_00.TcPOU
///EL2002 | 2-channel digital output terminal 24 V DC, 0.5 A
FUNCTION_BLOCK EL2002_v1_00
VAR_INPUT
	En: BOOL;
	bDo_1: BOOL;
	bDo_2: BOOL;
END_VAR
VAR_OUTPUT
	EnO: BOOL;
	bError: BOOL;
END_VAR
VAR
	Channel_1_Output AT %Q*: BOOL;
	Channel_2_Output AT %Q*: BOOL;
	WcState_WcState AT %I*: BOOL;
	InfoData_State AT %I*: UINT;
END_VAR

EnO:=En;

IF En AND (WcState_WcState OR InfoData_State<>16#8) THEN
	bError:=TRUE;
ELSE
	bError:=FALSE;
END_IF

IF En THEN
	IF bError=FALSE THEN
		Channel_1_Output:=bDo_1;
		Channel_2_Output:=bDo_2;
	END_IF
END_IF

END_FUNCTION_BLOCK

// ---- POUs/Hardware/EtherCAT_Terminals/Digital_Outputs/EL2042_v1_00.TcPOU
///EL2042 | 2-channel digital output terminal 24 V DC, 2 x 4 A/1 x 8 A
FUNCTION_BLOCK EL2042_v1_00
VAR_INPUT
	En: BOOL;
	bDo_1: BOOL;
	bDo_2: BOOL;
END_VAR
VAR_OUTPUT
	EnO: BOOL;
	bError: BOOL;
END_VAR
VAR
	Channel_1_Output AT %Q*: BOOL;
	Channel_2_Output AT %Q*: BOOL;
	WcState_WcState AT %I*: BOOL;
	InfoData_State AT %I*: UINT;
END_VAR

EnO:=En;

IF En AND (WcState_WcState OR InfoData_State<>16#8) THEN
	bError:=TRUE;
ELSE
	bError:=FALSE;
END_IF

IF En THEN
	IF bError=FALSE THEN
		Channel_1_Output:=bDo_1;
		Channel_2_Output:=bDo_2;
	END_IF
END_IF

END_FUNCTION_BLOCK

// ---- POUs/Hardware/EtherCAT_Terminals/Digital_Outputs/EL2124_v1_00.TcPOU
///EL2124 | 4-channel digital output terminal 5 V DC, 20 mA
FUNCTION_BLOCK EL2124_v1_00
VAR_INPUT
	En: BOOL;
	bDo_1: BOOL;
	bDo_2: BOOL;
	bDo_3: BOOL;
	bDo_4: BOOL;
END_VAR
VAR_OUTPUT
	EnO: BOOL;
	bError: BOOL;
END_VAR
VAR
	Channel_1_Output AT %Q*: BOOL;
	Channel_2_Output AT %Q*: BOOL;
	Channel_3_Output AT %Q*: BOOL;
	Channel_4_Output AT %Q*: BOOL;
	WcState_WcState AT %I*: BOOL;
	InfoData_State AT %I*: UINT;
END_VAR

EnO:=En;

IF En AND (WcState_WcState OR InfoData_State<>16#8) THEN
	bError:=TRUE;
ELSE
	bError:=FALSE;
END_IF

IF En THEN
	IF bError=FALSE THEN
		Channel_1_Output:=bDo_1;
		Channel_2_Output:=bDo_2;
		Channel_3_Output:=bDo_3;
		Channel_4_Output:=bDo_4;
	END_IF
END_IF

END_FUNCTION_BLOCK

// ---- POUs/Hardware/EtherCAT_Terminals/Digital_Outputs/EL2202_v0_00.TcPOU
///EL2202 | XFC, 2-channel digital output terminal 24 V DC, TON/TOFF 1 µs, push-pull outputs, tri-state
FUNCTION_BLOCK EL2202_v0_00

END_FUNCTION_BLOCK

// ---- POUs/Hardware/EtherCAT_Terminals/Digital_Outputs/EL2252_v0_00.TcPOU
///EL2252 | XFC, 2-channel digital output terminal with time stamp, tri-state
FUNCTION_BLOCK EL2252_v0_00

END_FUNCTION_BLOCK

// ---- POUs/Hardware/EtherCAT_Terminals/Digital_Outputs/EL2258_v0_00.TcPOU
///EL2258 | XFC, 8-channel digital output terminal with time stamp
FUNCTION_BLOCK EL2258_v0_00

END_FUNCTION_BLOCK

// ---- POUs/Hardware/EtherCAT_Terminals/Digital_Outputs/EL2262_v0_00.TcPOU
///EL2262 | XFC, 2-channel digital output terminal with oversampling
FUNCTION_BLOCK EL2262_v0_00

END_FUNCTION_BLOCK

// ---- POUs/Hardware/EtherCAT_Terminals/Digital_Outputs/EL2535_v0_00.TcPOU
///EL2535 | 2-channel pulse width current terminals 24 V DC
FUNCTION_BLOCK EL2535_v0_00

END_FUNCTION_BLOCK

// ---- POUs/Hardware/EtherCAT_Terminals/Digital_Outputs/FB_EL2008_v1_00.TcPOU
///EL2008 | 8-channel digital output terminal 24 V DC, 0.5 A
FUNCTION_BLOCK FB_EL2008_v1_00
VAR_INPUT
	En: BOOL;
	bDo_1: BOOL;
	bDo_2: BOOL;
	bDo_3: BOOL;
	bDo_4: BOOL;
	bDo_5: BOOL;
	bDo_6: BOOL;
	bDo_7: BOOL;
	bDo_8: BOOL;
END_VAR
VAR_OUTPUT
	EnO: BOOL;
	bError: BOOL;
END_VAR
VAR
	Channel_1_Output AT %Q*: BOOL;
	Channel_2_Output AT %Q*: BOOL;
	Channel_3_Output AT %Q*: BOOL;
	Channel_4_Output AT %Q*: BOOL;
	Channel_5_Output AT %Q*: BOOL;
	Channel_6_Output AT %Q*: BOOL;
	Channel_7_Output AT %Q*: BOOL;
	Channel_8_Output AT %Q*: BOOL;
	WcState_WcState AT %I*: BOOL;
	InfoData_State AT %I*: UINT;
END_VAR

EnO:=En;

IF En AND (WcState_WcState OR InfoData_State<>16#8) THEN
	bError:=TRUE;
ELSE
	bError:=FALSE;
END_IF

IF En THEN
	IF bError=FALSE THEN
		Channel_1_Output:=bDo_1;
		Channel_2_Output:=bDo_2;
		Channel_3_Output:=bDo_3;
		Channel_4_Output:=bDo_4;
		Channel_5_Output:=bDo_5;
		Channel_6_Output:=bDo_6;
		Channel_7_Output:=bDo_7;
		Channel_8_Output:=bDo_8;
	END_IF
END_IF

END_FUNCTION_BLOCK

// ---- POUs/Hardware/EtherCAT_Terminals/Digital_Outputs/Safety_Terminals/EL1904_v0_00.TcPOU
///EL1904 | 4-channel digital input terminal, TwinSAFE, 24 V DC
FUNCTION_BLOCK EL1904_v0_00

END_FUNCTION_BLOCK

// ---- POUs/Hardware/EtherCAT_Terminals/Digital_Outputs/Safety_Terminals/EL2901_v0_00.TcPOU
///EL2901 | Potential supply terminal, TwinSAFE, 24 V DC, 10 A
FUNCTION_BLOCK EL2901_v0_00

END_FUNCTION_BLOCK

// ---- POUs/Hardware/EtherCAT_Terminals/Digital_Outputs/Safety_Terminals/EL2902_v0_00.TcPOU
///EL2902 | 2-channel digital output terminal, TwinSAFE, 24 V DC, 2.3 A
FUNCTION_BLOCK EL2902_v0_00

END_FUNCTION_BLOCK

// ---- POUs/Hardware/EtherCAT_Terminals/Digital_Outputs/Safety_Terminals/FB_EL2904_v1_00.TcPOU
///EL2904 | 4-channel digital output terminal, TwinSAFE, 24 V DC, 0.5 A
FUNCTION_BLOCK FB_EL2904_v1_00
VAR_INPUT
	En: BOOL;
END_VAR
VAR_OUTPUT
	EnO: BOOL;
	bDo_1: BOOL;
	bDo_2: BOOL;
	bDo_3: BOOL;
	bDo_4: BOOL;
	bError: BOOL;
	sState: STRING;
	sDiag: STRING;
END_VAR
VAR
	Message_X_Info_Data_State AT %I*: USINT;
	Message_X_Info_Data_Diag AT %I*: USINT;
	Message_X_Output_Safe_Data AT %I*: BYTE;
	WcState_WcState AT %I*: BOOL;
	InfoData_State AT %I*: UINT;
END_VAR

EnO:=En;

IF En AND (WcState_WcState OR InfoData_State<>16#8) THEN
	bError:=TRUE;
ELSE
	bError:=FALSE;
END_IF

IF En THEN
	IF bError=FALSE THEN
		CASE Message_X_Info_Data_State OF
		0:
			sState:='Undefined';
		100:
			sState:='RESET';
		101:
			sState:='SESSION';
		102:
			sState:='CONNECTION';
		103:
			sState:='PARAMETER';
		104:
			sState:='DATA';
		105:
			sState:='SHUTDOWN';
		ELSE	
			sState:='Unknown';
		END_CASE

		sDiag:=USINT_TO_STRING(Message_X_Info_Data_Diag);

		bDo_1:=Message_X_Output_Safe_Data.0;
		bDo_2:=Message_X_Output_Safe_Data.1;
		bDo_3:=Message_X_Output_Safe_Data.2;
		bDo_4:=Message_X_Output_Safe_Data.3;
	ELSE
		sState:='';
		sDiag:='';

	END_IF
END_IF

END_FUNCTION_BLOCK

// ---- POUs/Hardware/EtherCAT_Terminals/Digital_Outputs/Safety_Terminals/FB_EL6900_v1_00.TcPOU
///EL6900 | TwinSAFE PLC
FUNCTION_BLOCK FB_EL6900_v1_00
VAR_INPUT
	En: BOOL;
END_VAR
VAR_OUTPUT
	EnO: BOOL;
	bError: BOOL;
END_VAR
VAR
	WcState_WcState AT %I*: BOOL;
	InfoData_State AT %I*: UINT;
END_VAR

EnO:=En;

IF En AND (WcState_WcState OR InfoData_State<>16#8) THEN
	bError:=TRUE;
ELSE
	bError:=FALSE;
END_IF

END_FUNCTION_BLOCK

// ---- POUs/Hardware/EtherCAT_Terminals/Motion/EL7211_v1_00.TcPOU
///EL7211 | Servo motor termional 5 A
FUNCTION_BLOCK EL7211_v1_00
VAR_INPUT
	En: BOOL;
END_VAR
VAR_OUTPUT
	EnO: BOOL;

	bError: BOOL;
END_VAR
VAR
	WcState_WcState AT %I*: BOOL;
	InfoData_State AT %I*: UINT;
END_VAR

EnO:=En;

IF En AND (WcState_WcState OR InfoData_State<>16#8) THEN
	bError:=TRUE;
ELSE
	bError:=FALSE;
END_IF

END_FUNCTION_BLOCK

// ---- POUs/Hardware/EtherCAT_Terminals/Motion/EL9576_v1_00.TcPOU
///EL9576 | Brake terminal (vap and resistor)
FUNCTION_BLOCK EL9576_v1_00
VAR_INPUT
	En: BOOL;
END_VAR
VAR_OUTPUT
	EnO: BOOL;
	bError: BOOL;	
	OverTemperature: BOOL;
	I2TError : BOOL;
	I2TWarning : BOOL;
	OverVoltage  : BOOL;
	UnderVoltage : BOOL;
	ChopperOn : BOOL;
	DCLinkVoltage : LREAL;
	DutyCycle  : LREAL;
	ResistorCurrent : LREAL;
	
END_VAR
VAR
	BCTOverTemperature AT %I*: BOOL;
	BCTI2TError AT %I*: BOOL;
	BCTI2TWarning AT %I*: BOOL;
	BCTOverVoltage  AT %I*: BOOL;
	BCTUnderVoltage  AT %I*: BOOL;
	BCTChopperOn  AT %I*: BOOL;
	BCTDCLinkVoltage AT %I*: UDINT;
	BCTDutyCycle  AT %I*: USINT;
	BCTResistorCurrent AT %I*: UDINT;
	WcState_WcState AT %I*: BOOL;
	InfoData_State AT %I*: UINT;
	
END_VAR

EnO:=En;

IF En AND (WcState_WcState OR InfoData_State<>16#8 OR BCTI2TError OR BCTI2TWarning OR BCTOverTemperature OR BCTOverVoltage OR BCTUnderVoltage) THEN
	bError:=TRUE;
ELSE
	bError:=FALSE;
END_IF

OverTemperature:=BCTOverTemperature;
I2TError:=BCTI2TError;
I2TWarning:=BCTI2TWarning;
OverVoltage:=BCTOverVoltage;
UnderVoltage:=bctUnderVoltage;
ChopperOn:=bctChopperOn;
DCLinkVoltage:=UDINT_TO_LREAL(bctDCLinkVoltage);
DutyCycle:=USINT_TO_LREAL(BCTDutyCycle);
ResistorCurrent:=UDINT_TO_LREAL(BCTResistorCurrent);

END_FUNCTION_BLOCK

// ---- POUs/Hardware/EtherCAT_Terminals/System/EL9505_V1_00.TcPOU
///EL9505 | 5v power supply treminal
FUNCTION_BLOCK EL9505_v1_00
VAR_INPUT
	En: BOOL;
END_VAR
VAR_OUTPUT
	EnO: BOOL;
	bError: BOOL;
END_VAR
VAR
	WcState_WcState AT %I*: BOOL;
	InfoData_State AT %I*: UINT;
END_VAR

EnO:=En;

IF En AND (WcState_WcState OR InfoData_State<>16#8) THEN
	bError:=TRUE;
ELSE
	bError:=FALSE;
END_IF

END_FUNCTION_BLOCK

// ---- POUs/Hardware/Other/EK1200.TcPOU
FUNCTION_BLOCK EK1200
VAR_INPUT
	En: BOOL;
END_VAR
VAR_OUTPUT
	EnO: BOOL;
END_VAR

EnO:=En;

END_FUNCTION_BLOCK

// ---- POUs/MAIN.TcPOU
PROGRAM MAIN
VAR
	sVersion: STRING:='1.0.0';
	M1:FB_DriveVirtual;
	M1Link:FB_NcAxis;
	bLimitFwd AT %I*: BOOL;
	bLimitBwd AT %I*: BOOL;
	bHomeSensor AT %I*: BOOL;
END_VAR

act();

ACTION ACT:
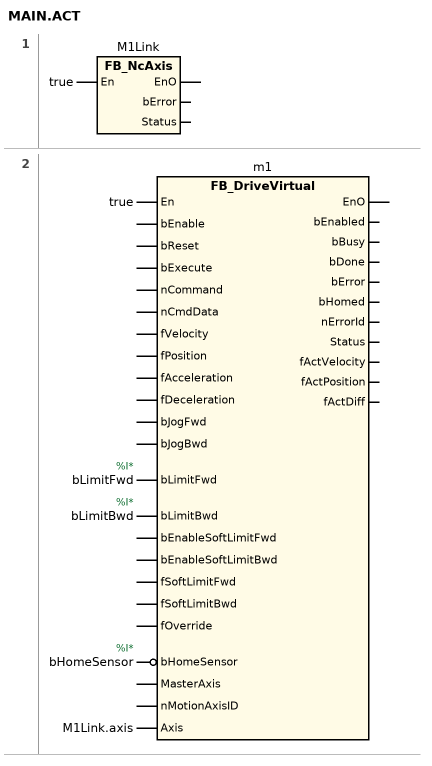
// NETWORK 1
M1Link(En := true); // FB_NcAxis

// NETWORK 2
//   bLimitFwd: AT %I*
//   bLimitBwd: AT %I*
//   bHomeSensor: AT %I*
m1(
    En := true,
    bLimitFwd := bLimitFwd,
    bLimitBwd := bLimitBwd,
    bHomeSensor := NOT bHomeSensor,
    Axis := M1Link.axis); // FB_DriveVirtual
END_ACTION

END_PROGRAM

// ---- POUs/Motion/FB_DriveVirtual.TcPOU
///#########################################################
///Function block to run a virtual drive with Nc
///	Library:		
///	Tc2_MC2.lib
///
///	Global Variables:
///	
///	Data types:
///	
///	External functions:
///
///###########################################################
FUNCTION_BLOCK FB_DriveVirtual
VAR
	sVersion: STRING:='1.0.2';
	bMovingRelOrAbs: BOOL;
END_VAR
VAR_INPUT
	En: BOOL;
	bEnable: BOOL;
	bReset: BOOL;
	bExecute: BOOL;
	/////	nCommand...
	/////	0 = Jog
	/////	1 = MoveVelocity
	/////	2 = MoveRelative
	/////	3 = MoveAbsolut
	/////	4 = MoveModulo
	/////	10 = Homing
	/////	20 = SuperInp >>>ToBe
	/////	30 = Gear
	nCommand: UINT;
	nCmdData: UINT;
	fVelocity: LREAL;
	fPosition: LREAL;
	fAcceleration: LREAL;
	fDeceleration: LREAL;
	bJogFwd: BOOL;
	bJogBwd: BOOL;
	bLimitFwd: BOOL;
	bLimitBwd: BOOL;	
	fOverride: LREAL := 100;
	bHomeSensor: BOOL;
	MasterAxis: AXIS_REF;
	nMotionAxisID:UDINT:=0;  //Axis id in Motion (NC) 
END_VAR
VAR_OUTPUT
	EnO: BOOL;
	bEnabled: BOOL;
	bBusy: BOOL;
	bDone: BOOL;
	bError: BOOL;
	bHomed: BOOL;
	nErrorId: UDINT;
	Status: ST_AxisStatus;
	fActVelocity: LREAL;
	fActPosition: LREAL;
	fActDiff: LREAL;

END_VAR
VAR_IN_OUT
	Axis: AXIS_REF;
END_VAR
VAR	
	bFirstScan: BOOL := TRUE;
	iCounter: INT := 0;
	fOldVelocity: LREAL;
	fbReset: MC_Reset;
	fbPower: MC_Power;
	fbHalt: MC_Halt;
	fbJog: MC_Jog;
	fbMoveVelocity: MC_MoveVelocity;
	fbMoveRelative: MC_MoveRelative;
	fbMoveAbsolute: MC_MoveAbsolute;
	fbMoveModulo: MC_MoveModulo;
	fbHome: MC_Home;
	fbGearInDyn: MC_GearInDyn;
	fbGearOut: MC_GearOut;
	stAxisStatus: DUT_AxisStatus_v0_01;
END_VAR

EnO:=En;

bHomed:=Axis.Status.Homed; //Add in DUT_AxisStatus later
bDone:=FALSE;

(*Reset*)
fbReset(
	Execute:=bReset AND Axis.Status.Error,
	Axis:=Axis,
	Done=> ,
	Busy=> ,
	Error=> ,
	ErrorID=> );

(*Power*)
fbPower(
	Axis:=Axis,
	Enable:=bEnable,
	Enable_Positive:=bLimitFwd AND bEnable,
	Enable_Negative:=bLimitBwd AND bEnable,
	Override:=fOverride,
	BufferMode:= ,
	Status=> ,
	Busy=> ,
	Active=> ,
	Error=> ,
	ErrorID=> );

(*Halt*)
fbHalt(
	Execute:=NOT bExecute  AND (((fbMoveVelocity.Busy OR fbPower.Busy) AND (nCommand=1)) OR (fbMoveRelative.Busy AND (nCommand=2)) OR (fbMoveAbsolute.Busy AND (nCommand=3)) OR (fbMoveModulo.Busy AND (nCommand=4)) OR (fbhome.Busy AND (nCommand=10))),
	Deceleration:=fDeceleration,
	Jerk:=0,
	BufferMode:= ,
	Options:= ,
	Axis:=Axis ,
	Done=> ,
	Busy=> ,
	Active=> ,
	CommandAborted=> ,
	Error=> ,
	ErrorID=> );

(*Jog (Command = 0)*)
fbJog(
	JogForward:=bJogFwd AND (nCommand=0) ,
	JogBackwards:=bJogBwd AND (nCommand=0) ,
	Mode:=nCmdData,
	Position:= ,
	Velocity:=fVelocity,
	Acceleration:=fAcceleration,
	Deceleration:=fDeceleration,
	Jerk:=0,
	Axis:=Axis,
	Done=> ,
	Busy=> ,
	Active=> ,
	CommandAborted=> ,
	Error=> ,
	ErrorID=> );

	;
	iCounter:=iCounter+1;
(*MoveVelocity (Command = 1)*)
fbMoveVelocity(
	Execute:=bExecute (*AND (fOldVelocity=fVelocity)*) AND (nCommand=1),
	Velocity:=ABS(fVelocity),
	Acceleration:=fAcceleration,
	Deceleration:=fDeceleration,
	Jerk:=0,
	Direction:=SEL(fVelocity<0, MC_Positive_Direction, MC_Negative_Direction),
	BufferMode:= ,
	Options:= ,
	Axis:=Axis,
	InVelocity=> ,
	Busy=> ,
	Active=> ,
	CommandAborted=> ,
	Error=> ,
	ErrorID=> );

(*MoveRelative (Command = 2)*)
fbMoveRelative(
	Execute:=bExecute AND (nCommand=2), 
	Distance:=fPosition, 
	Velocity:=ABS(fVelocity), 
	Acceleration:=fAcceleration,
	Deceleration:=fDeceleration,
	Jerk:=0,
	BufferMode:= , 
	Options:= , 
	Axis:=Axis, 
	Done=> , 
	Busy=> , 
	Active=> , 
	CommandAborted=> , 
	Error=> , 
	ErrorID=> );
	
IF nCommand=2 THEN
	bDone:=fbMoveRelative.Done;
END_IF
	
(*MoveAbsolute (Command = 3)*)
fbMoveAbsolute(
	Execute:=bExecute AND (nCommand=3),
	Position:=fPosition,
	Velocity:=ABS(fVelocity),
	Acceleration:=fAcceleration,
	Deceleration:=fDeceleration,
	Jerk:=0,
	BufferMode:= ,
	Options:= ,
	Axis:=Axis,
	Done=> ,
	Busy=> ,
	Active=> ,
	CommandAborted=> ,
	Error=> ,
	ErrorID=> );

IF nCommand=3 THEN
	bDone:=fbMoveAbsolute.Done;
END_IF

(*MoveModulo (Command = 4)*)
fbMoveModulo(
	Execute:=bExecute AND (nCommand=4), 
	Position:=fPosition, 
	Velocity:=ABS(fVelocity), 
	Acceleration:=fAcceleration, 
	Deceleration:=fDeceleration, 
	Jerk:=0, 
	Direction:=nCmdData, 
	BufferMode:= , 
	Options:= , 
	Axis:=Axis, 
	Done=> , 
	Busy=> , 
	Active=> , 
	CommandAborted=> , 
	Error=> , 
	ErrorID=> );

IF nCommand=4 THEN
	bDone:=fbMoveModulo.Done;
END_IF
	
(*Home (Command = 10)*)
fbHome(
	Execute:=bExecute AND (nCommand=10),
	Position:=fPosition,
	HomingMode:=nCmdData,
	BufferMode:= ,
	Options:= ,
	bCalibrationCam:=bHomeSensor,
	Axis:=Axis,
	Done=> ,
	Busy=> ,
	Active=> ,
	CommandAborted=> ,
	Error=> ,
	ErrorID=> );

IF nCommand=10 THEN
	bDone:=fbHome.Done;
END_IF

(*Gear (Command = 30)*)
fbGearInDyn(
	Enable:=bExecute  AND (nCommand=30),
	GearRatio:=SEL(nCmdData>0, 1,fVelocity), 
	Acceleration:=fAcceleration,
	Deceleration:=fDeceleration,
	Jerk:=0.0,
	BufferMode:= , 
	Options:= , 
	Master:=MasterAxis,
	Slave:=Axis,
	InGear=> , 
	Busy=> , 
	Active=> , 
	CommandAborted=> , 
	Error=> , 
	ErrorID=> );
	
fbGearOut(
	Execute:=NOT bExecute AND Axis.Status.NotMoving AND (nCommand=30),
	Slave:=Axis,
	Error=>,
	Done=>,
	ErrorID=>);


IF nCommand=30 THEN
	bDone:=Axis.Status.Coupled;
END_IF

fOldVelocity:=fVelocity;

(*Busy*)
bMovingRelOrAbs := (nCommand = 2 OR nCommand = 3) AND NOT axis.Status.InTargetPosition;
bBusy:=Axis.Status.HasJob OR Axis.Status.HomingBusy OR  bMovingRelOrAbs;

(*Enabled*)
bEnabled:=fbPower.Status;

(*Error from functions and Nc*)
IF fbPower.Error AND fbPower.Active THEN
	bError:=fbPower.Enable;
	nErrorId:=fbPower.ErrorID;
ELSIF fbHalt.Error AND fbHalt.Active THEN
	bError:=fbHalt.Execute;
	nErrorId:=fbHalt.ErrorID;
ELSIF fbJog.Error AND fbJog.Active THEN
	bError:=fbJog.JogForward OR fbJog.JogBackwards;
	nErrorId:=fbJog.ErrorID;
ELSIF fbMoveVelocity.Error AND fbMoveVelocity.Active THEN
	bError:=fbMoveVelocity.Execute;
	nErrorId:=fbMoveVelocity.ErrorID;
ELSIF fbMoveRelative.Error AND fbMoveRelative.Active THEN
	bError:=fbMoveRelative.Execute;
	nErrorId:=fbMoveRelative.ErrorID;
ELSIF fbMoveAbsolute.Error AND fbMoveAbsolute.Active THEN
	bError:=fbMoveAbsolute.Execute;
	nErrorId:=fbMoveAbsolute.ErrorID;
ELSIF fbMoveModulo.Error AND fbMoveModulo.Active THEN
	bError:=fbMoveModulo.Execute;
	nErrorId:=fbMoveModulo.ErrorID;
ELSIF fbHome.Error AND fbHome.Active THEN
	bError:=fbHome.Execute;
	nErrorId:=fbHome.ErrorID;
ELSIF fbGearInDyn.Error AND fbGearInDyn.Active THEN
	bError:=fbGearInDyn.Enable;
	nErrorId:=fbGearInDyn.ErrorID;
ELSIF fbGearOut.Error AND Axis.Status.Coupled THEN
	bError:=fbGearOut.Execute;
	nErrorId:=fbGearOut.ErrorID;
ELSIF Axis.Status.Error  THEN
	bError:=TRUE;
	nErrorId:=Axis.Status.ErrorID;
(*ELSIF fbWriteToNC.bError THEN
	bError:=TRUE;
	nErrorId:=fbWriteToNC.nErrorId;*)		
ELSE
	bError:=FALSE;
	nErrorId:=0;
END_IF;

(*Status from Nc*)
Status:=Axis.Status;

(*Axis id in motion "motor"*)
nMotionAxisID:=axis.NcToPlc.AxisId;

(*Actual Velocity*)
fActVelocity:=Axis.NcToPlc.ActVelo;

(*Actual Position*)
IF Axis.Status.OpMode.Modulo THEN
	fActPosition:=Axis.NcToPlc.ModuloActPos;
ELSE
	fActPosition:=Axis.NcToPlc.ActPos;
END_IF

(*Actual Position*)
fActDiff:=Axis.NcToPlc.PosDiff;


//Status struct for EPICS communication
stAxisStatus.bEnable:=bEnable;
stAxisStatus.bEnabled:=bEnabled;
stAxisStatus.bError:=bError;
stAxisStatus.bExecute:=bExecute;
stAxisStatus.bHomeSensor:=bHomeSensor;
stAxisStatus.bJogBwd:=bJogBwd;
stAxisStatus.bJogFwd:=bJogFwd;
stAxisStatus.bLimitBwd:=bLimitBwd;
stAxisStatus.bLimitFwd:=bLimitFwd;
stAxisStatus.bReset:=bReset;
stAxisStatus.fAcceleration:=fAcceleration;
stAxisStatus.fActDiff:=fActDiff;
stAxisStatus.fActPosition:=fActPosition;
stAxisStatus.fActVelocity:=fActVelocity;
stAxisStatus.fDeceleration:=fDeceleration;
stAxisStatus.fOverride:=fOverride;
stAxisStatus.fPosition:=fPosition;
stAxisStatus.fVelocity:=fVelocity;
stAxisStatus.nCmdData:=nCmdData;
stAxisStatus.nCommand:=nCommand;
stAxisStatus.nErrorId:=nErrorId;
stAxisStatus.bBusy:=bBusy;
stAxisStatus.bHomed:=bHomed;

IF bFirstScan THEN
	bFirstScan:=FALSE;
END_IF

END_FUNCTION_BLOCK
